(* CODESYS project Warehouse_Final_Plc.project
   Company: ifm electronic
   Description: Project template with CR711S configured 2.25MByte Standard 2.25MByte Safety
   Title: ifmCR711S_TemplateProject
   Version: 2.4.10.0

Project tree, tasks and I/O mapping:
  StandardPLC : CR711S Standard, ifm electronic, order no. CR711S, version 3.2.0.0
    application Application
      libraries: ifmR360-3, 1.1.1.0 (ifm electronic); Util, * (System); Standard, * (System); CR711S IOWrapper, 1.0.4.9 (ifm electronic); CAA CiA 405, 3.5.8.0 (CAA Technical Workgroup)
      task Task (cyclic, interval t#10ms, priority 0) calls PLC_PRG
      global variables inc1
      EVC
      program CR711S_Config [ST]: config_outputs, config_outgroups, config_inputs
      trace Trace (task Task): PLC_PRG.iSlopeLat, PLC_PRG.iSlopeLong
      program PLC_PRG [ST]
      visualisation Visualization
      program Inclination_logic [ST]
      program Temp_Logic [ST]
      program CAN_INIT [ST]
      program CAN_TX [FBD]
      trace Trace_1 (task ): Temp_Logic.TEMPval
      visualisation Visualization_1
      program test [FBD]
    HMI : HMI, ifm electronic, version 3.2.0.0
      User_LEDs : User_LEDs, ifm electronic, version 3.2.0.0
          input  UserLED0_I : LED_IEC_B_INPUT_MAPPING_TYPE  // UserLED0_I
          input  UserLED1_I : LED_IEC_B_INPUT_MAPPING_TYPE  // UserLED1_I
          input  UserLED2_I : LED_IEC_B_INPUT_MAPPING_TYPE  // UserLED2_I
          input  UserLED3_I : LED_IEC_B_INPUT_MAPPING_TYPE  // UserLED3_I
          output UserLED0_Q : LED_IEC_B_OUTPUT_MAPPING_TYPE  // User LED 0
          output UserLED1_Q : LED_IEC_B_OUTPUT_MAPPING_TYPE  // User LED 1
          output UserLED2_Q : LED_IEC_B_OUTPUT_MAPPING_TYPE  // User LED 2
          output UserLED3_Q : LED_IEC_B_OUTPUT_MAPPING_TYPE  // User LED 3
    Local_IO : Local_IO, ifm electronic, version 3.2.0.0
      System_Inputs : System_Inputs, ifm electronic, version 3.2.0.0
          input  VBB30 : IN_SYSTEM_VOLTAGE_INPUT_MAPPING_TYPE  // VBB30
          input  VBB15 : IN_SYSTEM_VOLTAGE_INPUT_MAPPING_TYPE  // VBB15
          input  TemperatureBoard0 : IN_TEMPERATURE_INPUT_MAPPING_TYPE  // TemperatureBoard0
          input  TemperatureChip0 : IN_TEMPERATURE_INPUT_MAPPING_TYPE  // TemperatureChip0
      Inputs : Inputs, ifm electronic, version 3.2.0.0
          input  IN0100_I : IN_MULTIFUNCTION_A_INPUT_MAPPING_TYPE  // IN0100_I
          input  IN0101_I : IN_MULTIFUNCTION_A_INPUT_MAPPING_TYPE  // IN0101_I
          input  IN0102_I : IN_MULTIFUNCTION_A_INPUT_MAPPING_TYPE  // IN0102_I
          input  IN0103_I : IN_MULTIFUNCTION_A_INPUT_MAPPING_TYPE  // IN0103_I
          input  IN0200_I : IN_MULTIFUNCTION_A_INPUT_MAPPING_TYPE  // IN0200_I
          input  IN0201_I : IN_MULTIFUNCTION_A_INPUT_MAPPING_TYPE  // IN0201_I
          input  IN0202_I : IN_MULTIFUNCTION_A_INPUT_MAPPING_TYPE  // IN0202_I
          input  IN0203_I : IN_MULTIFUNCTION_A_INPUT_MAPPING_TYPE  // IN0203_I
          input  IN0600_I : IN_MULTIFUNCTION_A_INPUT_MAPPING_TYPE  // IN0600_I
          input  IN0601_I : IN_MULTIFUNCTION_A_INPUT_MAPPING_TYPE  // IN0601_I
          input  IN0602_I : IN_MULTIFUNCTION_A_INPUT_MAPPING_TYPE  // IN0602_I
          input  IN0603_I : IN_MULTIFUNCTION_A_INPUT_MAPPING_TYPE  // IN0603_I
          input  IN0700_I : IN_MULTIFUNCTION_A_INPUT_MAPPING_TYPE  // IN0700_I
          input  IN0701_I : IN_MULTIFUNCTION_A_INPUT_MAPPING_TYPE  // IN0701_I
          input  IN0702_I : IN_MULTIFUNCTION_A_INPUT_MAPPING_TYPE  // IN0702_I
          input  IN0703_I : IN_MULTIFUNCTION_A_INPUT_MAPPING_TYPE  // IN0703_I
          input  IN0400_I : IN_RESISTOR_A_INPUT_MAPPING_TYPE  // IN0400_I
          input  IN0401_I : IN_RESISTOR_A_INPUT_MAPPING_TYPE  // IN0401_I
          input  IN0900_I : IN_RESISTOR_A_INPUT_MAPPING_TYPE  // IN0900_I
          input  IN0901_I : IN_RESISTOR_A_INPUT_MAPPING_TYPE  // IN0901_I
          input  IN0300_I : IN_DIGITAL_B_INPUT_MAPPING_TYPE  // IN0300_I
          input  IN0301_I : IN_DIGITAL_B_INPUT_MAPPING_TYPE  // IN0301_I
          input  IN0800_I : IN_DIGITAL_B_INPUT_MAPPING_TYPE  // IN0800_I
          input  IN0801_I : IN_DIGITAL_B_INPUT_MAPPING_TYPE  // IN0801_I
          input  COM_RESET_I : IN_COMMUNICATION_RESET_INPUT_MAPPING_TYPE  // COM_RESET_I
          input  IN0000_I : IN_FREQUENCY_B_CHANNEL_A_INPUT_MAPPING_TYPE  // IN0000_I
          input  IN0002_I : IN_FREQUENCY_B_CHANNEL_A_INPUT_MAPPING_TYPE  // IN0002_I
          input  IN0500_I : IN_FREQUENCY_B_CHANNEL_A_INPUT_MAPPING_TYPE  // IN0500_I
          input  IN0502_I : IN_FREQUENCY_B_CHANNEL_A_INPUT_MAPPING_TYPE  // IN0502_I
          input  IN0001_I : IN_FREQUENCY_B_CHANNEL_B_INPUT_MAPPING_TYPE  // IN0001_I
          input  IN0003_I : IN_FREQUENCY_B_CHANNEL_B_INPUT_MAPPING_TYPE  // IN0003_I
          input  IN0501_I : IN_FREQUENCY_B_CHANNEL_B_INPUT_MAPPING_TYPE  // IN0501_I
          input  IN0503_I : IN_FREQUENCY_B_CHANNEL_B_INPUT_MAPPING_TYPE  // IN0503_I
      Outputs : Outputs, ifm electronic, version 3.2.0.0
          input  OUT0006_I : OUT_PWM_40_BRIDGE_A_INPUT_MAPPING_TYPE  // OUT0006_I
          input  OUT0106_I : OUT_PWM_40_BRIDGE_A_INPUT_MAPPING_TYPE  // OUT0106_I
          input  OUT0206_I : OUT_PWM_40_BRIDGE_A_INPUT_MAPPING_TYPE  // OUT0206_I
          input  OUT0008_I : OUT_PWM_40_A_INPUT_MAPPING_TYPE  // OUT0008_I
          input  OUT0108_I : OUT_PWM_40_A_INPUT_MAPPING_TYPE  // OUT0108_I
          input  OUT0208_I : OUT_PWM_40_A_INPUT_MAPPING_TYPE  // OUT0208_I
          input  OUT0000_I : OUT_PWM_25_A_INPUT_MAPPING_TYPE  // OUT0000_I
          input  OUT0002_I : OUT_PWM_25_A_INPUT_MAPPING_TYPE  // OUT0002_I
          input  OUT0004_I : OUT_PWM_25_A_INPUT_MAPPING_TYPE  // OUT0004_I
          input  OUT0100_I : OUT_PWM_25_A_INPUT_MAPPING_TYPE  // OUT0100_I
          input  OUT0102_I : OUT_PWM_25_A_INPUT_MAPPING_TYPE  // OUT0102_I
          input  OUT0104_I : OUT_PWM_25_A_INPUT_MAPPING_TYPE  // OUT0104_I
          input  OUT0200_I : OUT_PWM_25_A_INPUT_MAPPING_TYPE  // OUT0200_I
          input  OUT0202_I : OUT_PWM_25_A_INPUT_MAPPING_TYPE  // OUT0202_I
          input  OUT0204_I : OUT_PWM_25_A_INPUT_MAPPING_TYPE  // OUT0204_I
          input  OUT3001_I : OUT_VOLTAGE_A_INPUT_MAPPING_TYPE  // OUT3001_I
          input  OUT3000_I : OUT_SUPPLY_A_INPUT_MAPPING_TYPE  // OUT3000_I
          input  OUT0001_I : OUT_PWM_25_B_INPUT_MAPPING_TYPE  // OUT0001_I
          input  OUT0003_I : OUT_PWM_25_B_INPUT_MAPPING_TYPE  // OUT0003_I
          input  OUT0005_I : OUT_PWM_25_B_INPUT_MAPPING_TYPE  // OUT0005_I
          input  OUT0101_I : OUT_PWM_25_B_INPUT_MAPPING_TYPE  // OUT0101_I
          input  OUT0103_I : OUT_PWM_25_B_INPUT_MAPPING_TYPE  // OUT0103_I
          input  OUT0105_I : OUT_PWM_25_B_INPUT_MAPPING_TYPE  // OUT0105_I
          input  OUT0201_I : OUT_PWM_25_B_INPUT_MAPPING_TYPE  // OUT0201_I
          input  OUT0203_I : OUT_PWM_25_B_INPUT_MAPPING_TYPE  // OUT0203_I
          input  OUT0205_I : OUT_PWM_25_B_INPUT_MAPPING_TYPE  // OUT0205_I
          input  OUT0007_I : OUT_PWM_40_BRIDGE_A_INPUT_MAPPING_TYPE  // OUT0007_I
          input  OUT0107_I : OUT_PWM_40_BRIDGE_A_INPUT_MAPPING_TYPE  // OUT0107_I
          input  OUT0207_I : OUT_PWM_40_BRIDGE_A_INPUT_MAPPING_TYPE  // OUT0207_I
          output OUT0006_Q : OUT_PWM_40_BRIDGE_A_OUTPUT_MAPPING_TYPE  // OUT0006_Q
          output OUT0106_Q : OUT_PWM_40_BRIDGE_A_OUTPUT_MAPPING_TYPE  // OUT0106_Q
          output OUT0206_Q : OUT_PWM_40_BRIDGE_A_OUTPUT_MAPPING_TYPE  // OUT0206_Q
          output OUT0008_Q : OUT_PWM_40_A_OUTPUT_MAPPING_TYPE  // OUT0008_Q
          output OUT0108_Q : OUT_PWM_40_A_OUTPUT_MAPPING_TYPE  // OUT0108_Q
          output OUT0208_Q : OUT_PWM_40_A_OUTPUT_MAPPING_TYPE  // OUT0208_Q
          output OUT0000_Q : OUT_PWM_25_A_OUTPUT_MAPPING_TYPE  // OUT0000_Q
          output OUT0002_Q : OUT_PWM_25_A_OUTPUT_MAPPING_TYPE  // OUT0002_Q
          output OUT0004_Q : OUT_PWM_25_A_OUTPUT_MAPPING_TYPE  // OUT0004_Q
          output OUT0100_Q : OUT_PWM_25_A_OUTPUT_MAPPING_TYPE  // OUT0100_Q
          output OUT0102_Q : OUT_PWM_25_A_OUTPUT_MAPPING_TYPE  // OUT0102_Q
          output OUT0104_Q : OUT_PWM_25_A_OUTPUT_MAPPING_TYPE  // OUT0104_Q
          output OUT0200_Q : OUT_PWM_25_A_OUTPUT_MAPPING_TYPE  // OUT0200_Q
          output OUT0202_Q : OUT_PWM_25_A_OUTPUT_MAPPING_TYPE  // OUT0202_Q
          output OUT0204_Q : OUT_PWM_25_A_OUTPUT_MAPPING_TYPE  // OUT0204_Q
          output OUT3001_Q : OUT_VOLTAGE_A_OUTPUT_MAPPING_TYPE  // OUT3001_Q
          output OUT3000_Q : OUT_SUPPLY_A_OUTPUT_MAPPING_TYPE  // OUT3000_Q
          output OUT0001_Q : OUT_PWM_25_B_OUTPUT_MAPPING_TYPE  // OUT0001_Q
          output OUT0003_Q : OUT_PWM_25_B_OUTPUT_MAPPING_TYPE  // OUT0003_Q
          output OUT0005_Q : OUT_PWM_25_B_OUTPUT_MAPPING_TYPE  // OUT0005_Q
          output OUT0101_Q : OUT_PWM_25_B_OUTPUT_MAPPING_TYPE  // OUT0101_Q
          output OUT0103_Q : OUT_PWM_25_B_OUTPUT_MAPPING_TYPE  // OUT0103_Q
          output OUT0105_Q : OUT_PWM_25_B_OUTPUT_MAPPING_TYPE  // OUT0105_Q
          output OUT0201_Q : OUT_PWM_25_B_OUTPUT_MAPPING_TYPE  // OUT0201_Q
          output OUT0203_Q : OUT_PWM_25_B_OUTPUT_MAPPING_TYPE  // OUT0203_Q
          output OUT0205_Q : OUT_PWM_25_B_OUTPUT_MAPPING_TYPE  // OUT0205_Q
          output OUT0007_Q : OUT_PWM_40_BRIDGE_A_OUTPUT_MAPPING_TYPE  // OUT0007_Q
          output OUT0107_Q : OUT_PWM_40_BRIDGE_A_OUTPUT_MAPPING_TYPE  // OUT0107_Q
          output OUT0207_Q : OUT_PWM_40_BRIDGE_A_OUTPUT_MAPPING_TYPE  // OUT0207_Q
      System_Outputs : System_Outputs, ifm electronic, version 3.2.0.0
          input  VBB0_SW_I : OUT_GROUP_SWITCH_INPUT_MAPPING_TYPE  // VBB0_SW_I
          input  VBB1_SW_I : OUT_GROUP_SWITCH_INPUT_MAPPING_TYPE  // VBB1_SW_I
          input  VBB2_SW_I : OUT_GROUP_SWITCH_INPUT_MAPPING_TYPE  // VBB2_SW_I
          output VBB0_SW_Q : OUT_GROUP_SWITCH_OUTPUT_MAPPING_TYPE  // VBB0_SW_Q
          output VBB1_SW_Q : OUT_GROUP_SWITCH_OUTPUT_MAPPING_TYPE  // VBB1_SW_Q
          output VBB2_SW_Q : OUT_GROUP_SWITCH_OUTPUT_MAPPING_TYPE  // VBB2_SW_Q
          output SUPPLY_SWITCH_Q : OUT_SYS_SWITCH_OUTPUT_MAPPING_TYPE  // SUPPLY_SWITCH_Q
    Communication : Communication, ifm electronic, version 3.2.0.0
      CAN : CAN, ifm electronic, version 3.2.0.0
        CANbus : CANbus, ifm electronic, version 1.0.1.1
          CANopen_Manager : CANopen_Manager, 3S - Smart Software Solutions GmbH, version 3.5.16.0
              settings: NMT Start All = TRUE; ConfigVersion = 50659584
            JN2100 : JN2100, ifm electornic GmbH, order no. JN2100, version Revision=16#000000AA, FileVersion=1.1, File=JN2100_V2.5.4.eds
                settings: General Options.Optional Device = TRUE; General Options.Reset Node = FALSE; NODEIDSAVED = 10; SDO Timeout = 1000000; PDO_Autoconfig = FALSE; EXPERTSETTINGS = True; Emergency-General Parameters.Emergency COBID = 16#0000008A; Heartbeat-Producer Time = 200; PDO 16#1800.COBID = 16#0000018A; PDO 16#1800.Transmission Type = 16#FE; PDO 16#1800.Event Timer = 50; Process by CANopenManager = TRUE; PDO 16#1801.COBID = 16#0000028A; PDO 16#1801.Transmission Type = 16#01; Process by CANopenManager = TRUE; PDO 16#1802.COBID = 16#0000038A; PDO 16#1802.Transmission Type = 16#01; Process by CANopenManager = TRUE; PDO 16#1803.COBID = 16#0000048A; Process by CANopenManager = TRUE; Slope long16.Subindex = 16#00; Slope lateral16.Subindex = 16#00; Slope long32.Subindex = 16#00; Slope lateral32.Subindex = 16#00; v effektive vector magnitude.Subindex = 16#00; a peak vector magnitude.Subindex = 16#00; a x vector.Subindex = 16#00; a y vector.Subindex = 16#00; a z vector.Subindex = 16#00; SDO List.Set Guardtime.Index = 16#100C; SDO List.Set Guardtime.Subindex = 16#00; SDO List.Set Guardtime.Value = 16#00000000; SDO List.Set Guardtime.Size = 16; SDO List.Set Guardtime.AbortIfError = FALSE; SDO List.Set Guardtime.JumpToLine = FALSE; SDO List.Set Guardtime.Line = 0; SDO List.Set Lifetime.Index = 16#100D; SDO List.Set Lifetime.Subindex = 16#00; SDO List.Set Lifetime.Value = 16#00000000; SDO List.Set Lifetime.Size = 8;
                  SDO List.Set Lifetime.AbortIfError = FALSE; SDO List.Set Lifetime.JumpToLine = FALSE; SDO List.Set Lifetime.Line = 0; SDO List.Set Heartbeat Producer.Index = 16#1017; SDO List.Set Heartbeat Producer.Subindex = 16#00; SDO List.Set Heartbeat Producer.Value = 16#000000C8; SDO List.Set Heartbeat Producer.Size = 16; SDO List.Set Heartbeat Producer.AbortIfError = FALSE; SDO List.Set Heartbeat Producer.JumpToLine = FALSE; SDO List.Set Heartbeat Producer.Line = 0; SDO List.Disable PDO.Index = 16#1800; SDO List.Disable PDO.Subindex = 16#01; SDO List.Disable PDO.Value = 16#8000018A; SDO List.Disable PDO.Size = 32; SDO List.Disable PDO.AbortIfError = FALSE; SDO List.Disable PDO.JumpToLine = FALSE; SDO List.Disable PDO.Line = 0; SDO List.Set transmission type.Index = 16#1800; SDO List.Set transmission type.Subindex = 16#02; SDO List.Set transmission type.Value = 16#FE; SDO List.Set transmission type.Size = 8; SDO List.Set transmission type.AbortIfError = FALSE; SDO List.Set transmission type.JumpToLine = FALSE; SDO List.Set transmission type.Line = 0; SDO List.Set inhibit time.Index = 16#1800; SDO List.Set inhibit time.Subindex = 16#03; SDO List.Set inhibit time.Value = 16#0000; SDO List.Set inhibit time.Size = 16; SDO List.Set inhibit time.AbortIfError = FALSE; SDO List.Set inhibit time.JumpToLine = FALSE; SDO List.Set inhibit time.Line = 0; SDO List.Set event time.Index = 16#1800; SDO List.Set event time.Subindex = 16#05; SDO List.Set event time.Value = 16#0032; SDO List.Set event time.Size = 16; SDO List.Set event time.AbortIfError = FALSE; SDO List.Set event time.JumpToLine = FALSE; SDO List.Set event time.Line = 0; SDO List.Clear pdo mapping.Index = 16#1A00; SDO List.Clear pdo mapping.Subindex = 16#00;
                  SDO List.Clear pdo mapping.Value = 16#0; SDO List.Clear pdo mapping.Size = 8; SDO List.Clear pdo mapping.AbortIfError = FALSE; SDO List.Clear pdo mapping.JumpToLine = FALSE; SDO List.Clear pdo mapping.Line = 0; SDO List.Set Mapping.Index = 16#1A00; SDO List.Set Mapping.Subindex = 16#01; SDO List.Set Mapping.Value = 16#60100010; SDO List.Set Mapping.Size = 32; SDO List.Set Mapping.AbortIfError = FALSE; SDO List.Set Mapping.JumpToLine = FALSE; SDO List.Set Mapping.Line = 0; SDO List.Set Mapping.Index = 16#1A00; SDO List.Set Mapping.Subindex = 16#02; SDO List.Set Mapping.Value = 16#60200010; SDO List.Set Mapping.Size = 32; SDO List.Set Mapping.AbortIfError = FALSE; SDO List.Set Mapping.JumpToLine = FALSE; SDO List.Set Mapping.Line = 0; SDO List.Set number of mappings.Index = 16#1A00; SDO List.Set number of mappings.Subindex = 16#00; SDO List.Set number of mappings.Value = 16#02; SDO List.Set number of mappings.Size = 8; SDO List.Set number of mappings.AbortIfError = FALSE; SDO List.Set number of mappings.JumpToLine = FALSE; SDO List.Set number of mappings.Line = 0; SDO List.Set and enable COB-ID.Index = 16#1800; SDO List.Set and enable COB-ID.Subindex = 16#01; SDO List.Set and enable COB-ID.Value = 16#0000018A; SDO List.Set and enable COB-ID.Size = 32; SDO List.Set and enable COB-ID.AbortIfError = FALSE; SDO List.Set and enable COB-ID.JumpToLine = FALSE; SDO List.Set and enable COB-ID.Line = 0; SDO List.Disable PDO.Index = 16#1801; SDO List.Disable PDO.Subindex = 16#01; SDO List.Disable PDO.Value = 16#8000028A; SDO List.Disable PDO.Size = 32; SDO List.Disable PDO.AbortIfError = FALSE; SDO List.Disable PDO.JumpToLine = FALSE; SDO List.Disable PDO.Line = 0;
                  SDO List.Set transmission type.Index = 16#1801; SDO List.Set transmission type.Subindex = 16#02; SDO List.Set transmission type.Value = 16#01; SDO List.Set transmission type.Size = 8; SDO List.Set transmission type.AbortIfError = FALSE; SDO List.Set transmission type.JumpToLine = FALSE; SDO List.Set transmission type.Line = 0; SDO List.Set inhibit time.Index = 16#1801; SDO List.Set inhibit time.Subindex = 16#03; SDO List.Set inhibit time.Value = 16#0000; SDO List.Set inhibit time.Size = 16; SDO List.Set inhibit time.AbortIfError = FALSE; SDO List.Set inhibit time.JumpToLine = FALSE; SDO List.Set inhibit time.Line = 0; SDO List.Set event time.Index = 16#1801; SDO List.Set event time.Subindex = 16#05; SDO List.Set event time.Value = 16#000A; SDO List.Set event time.Size = 16; SDO List.Set event time.AbortIfError = FALSE; SDO List.Set event time.JumpToLine = FALSE; SDO List.Set event time.Line = 0; SDO List.Clear pdo mapping.Index = 16#1A01; SDO List.Clear pdo mapping.Subindex = 16#00; SDO List.Clear pdo mapping.Value = 16#0; SDO List.Clear pdo mapping.Size = 8; SDO List.Clear pdo mapping.AbortIfError = FALSE; SDO List.Clear pdo mapping.JumpToLine = FALSE; SDO List.Clear pdo mapping.Line = 0; SDO List.Set Mapping.Index = 16#1A01; SDO List.Set Mapping.Subindex = 16#01; SDO List.Set Mapping.Value = 16#61100020; SDO List.Set Mapping.Size = 32; SDO List.Set Mapping.AbortIfError = FALSE; SDO List.Set Mapping.JumpToLine = FALSE; SDO List.Set Mapping.Line = 0; SDO List.Set Mapping.Index = 16#1A01; SDO List.Set Mapping.Subindex = 16#02; SDO List.Set Mapping.Value = 16#61200020; SDO List.Set Mapping.Size = 32; SDO List.Set Mapping.AbortIfError = FALSE;
                  SDO List.Set Mapping.JumpToLine = FALSE; SDO List.Set Mapping.Line = 0; SDO List.Set number of mappings.Index = 16#1A01; SDO List.Set number of mappings.Subindex = 16#00; SDO List.Set number of mappings.Value = 16#02; SDO List.Set number of mappings.Size = 8; SDO List.Set number of mappings.AbortIfError = FALSE; SDO List.Set number of mappings.JumpToLine = FALSE; SDO List.Set number of mappings.Line = 0; SDO List.Set and enable COB-ID.Index = 16#1801; SDO List.Set and enable COB-ID.Subindex = 16#01; SDO List.Set and enable COB-ID.Value = 16#0000028A; SDO List.Set and enable COB-ID.Size = 32; SDO List.Set and enable COB-ID.AbortIfError = FALSE; SDO List.Set and enable COB-ID.JumpToLine = FALSE; SDO List.Set and enable COB-ID.Line = 0; SDO List.Disable PDO.Index = 16#1802; SDO List.Disable PDO.Subindex = 16#01; SDO List.Disable PDO.Value = 16#8000038A; SDO List.Disable PDO.Size = 32; SDO List.Disable PDO.AbortIfError = FALSE; SDO List.Disable PDO.JumpToLine = FALSE; SDO List.Disable PDO.Line = 0; SDO List.Set transmission type.Index = 16#1802; SDO List.Set transmission type.Subindex = 16#02; SDO List.Set transmission type.Value = 16#01; SDO List.Set transmission type.Size = 8; SDO List.Set transmission type.AbortIfError = FALSE; SDO List.Set transmission type.JumpToLine = FALSE; SDO List.Set transmission type.Line = 0; SDO List.Set inhibit time.Index = 16#1802; SDO List.Set inhibit time.Subindex = 16#03; SDO List.Set inhibit time.Value = 16#0000; SDO List.Set inhibit time.Size = 16; SDO List.Set inhibit time.AbortIfError = FALSE; SDO List.Set inhibit time.JumpToLine = FALSE; SDO List.Set inhibit time.Line = 0; SDO List.Set event time.Index = 16#1802; SDO List.Set event time.Subindex = 16#05; SDO List.Set event time.Value = 16#000A;
                  SDO List.Set event time.Size = 16; SDO List.Set event time.AbortIfError = FALSE; SDO List.Set event time.JumpToLine = FALSE; SDO List.Set event time.Line = 0; SDO List.Clear pdo mapping.Index = 16#1A02; SDO List.Clear pdo mapping.Subindex = 16#00; SDO List.Clear pdo mapping.Value = 16#0; SDO List.Clear pdo mapping.Size = 8; SDO List.Clear pdo mapping.AbortIfError = FALSE; SDO List.Clear pdo mapping.JumpToLine = FALSE; SDO List.Clear pdo mapping.Line = 0; SDO List.Set Mapping.Index = 16#1A02; SDO List.Set Mapping.Subindex = 16#01; SDO List.Set Mapping.Value = 16#5C100020; SDO List.Set Mapping.Size = 32; SDO List.Set Mapping.AbortIfError = FALSE; SDO List.Set Mapping.JumpToLine = FALSE; SDO List.Set Mapping.Line = 0; SDO List.Set Mapping.Index = 16#1A02; SDO List.Set Mapping.Subindex = 16#02; SDO List.Set Mapping.Value = 16#5C110020; SDO List.Set Mapping.Size = 32; SDO List.Set Mapping.AbortIfError = FALSE; SDO List.Set Mapping.JumpToLine = FALSE; SDO List.Set Mapping.Line = 0; SDO List.Set number of mappings.Index = 16#1A02; SDO List.Set number of mappings.Subindex = 16#00; SDO List.Set number of mappings.Value = 16#02; SDO List.Set number of mappings.Size = 8; SDO List.Set number of mappings.AbortIfError = FALSE; SDO List.Set number of mappings.JumpToLine = FALSE; SDO List.Set number of mappings.Line = 0; SDO List.Set and enable COB-ID.Index = 16#1802; SDO List.Set and enable COB-ID.Subindex = 16#01; SDO List.Set and enable COB-ID.Value = 16#0000038A; SDO List.Set and enable COB-ID.Size = 32; SDO List.Set and enable COB-ID.AbortIfError = FALSE; SDO List.Set and enable COB-ID.JumpToLine = FALSE; SDO List.Set and enable COB-ID.Line = 0; SDO List.Disable PDO.Index = 16#1803;
                  SDO List.Disable PDO.Subindex = 16#01; SDO List.Disable PDO.Value = 16#8000048A; SDO List.Disable PDO.Size = 32; SDO List.Disable PDO.AbortIfError = FALSE; SDO List.Disable PDO.JumpToLine = FALSE; SDO List.Disable PDO.Line = 0; SDO List.Set transmission type.Index = 16#1803; SDO List.Set transmission type.Subindex = 16#02; SDO List.Set transmission type.Value = 16#FF; SDO List.Set transmission type.Size = 8; SDO List.Set transmission type.AbortIfError = FALSE; SDO List.Set transmission type.JumpToLine = FALSE; SDO List.Set transmission type.Line = 0; SDO List.Set inhibit time.Index = 16#1803; SDO List.Set inhibit time.Subindex = 16#03; SDO List.Set inhibit time.Value = 16#0000; SDO List.Set inhibit time.Size = 16; SDO List.Set inhibit time.AbortIfError = FALSE; SDO List.Set inhibit time.JumpToLine = FALSE; SDO List.Set inhibit time.Line = 0; SDO List.Set event time.Index = 16#1803; SDO List.Set event time.Subindex = 16#05; SDO List.Set event time.Value = 16#000A; SDO List.Set event time.Size = 16; SDO List.Set event time.AbortIfError = FALSE; SDO List.Set event time.JumpToLine = FALSE; SDO List.Set event time.Line = 0; SDO List.Clear pdo mapping.Index = 16#1A03; SDO List.Clear pdo mapping.Subindex = 16#00; SDO List.Clear pdo mapping.Value = 16#0; SDO List.Clear pdo mapping.Size = 8; SDO List.Clear pdo mapping.AbortIfError = FALSE; SDO List.Clear pdo mapping.JumpToLine = FALSE; SDO List.Clear pdo mapping.Line = 0; SDO List.Set Mapping.Index = 16#1A03; SDO List.Set Mapping.Subindex = 16#01; SDO List.Set Mapping.Value = 16#5D100010; SDO List.Set Mapping.Size = 32; SDO List.Set Mapping.AbortIfError = FALSE; SDO List.Set Mapping.JumpToLine = FALSE;
                  SDO List.Set Mapping.Line = 0; SDO List.Set Mapping.Index = 16#1A03; SDO List.Set Mapping.Subindex = 16#02; SDO List.Set Mapping.Value = 16#5D110010; SDO List.Set Mapping.Size = 32; SDO List.Set Mapping.AbortIfError = FALSE; SDO List.Set Mapping.JumpToLine = FALSE; SDO List.Set Mapping.Line = 0; SDO List.Set Mapping.Index = 16#1A03; SDO List.Set Mapping.Subindex = 16#03; SDO List.Set Mapping.Value = 16#5D120010; SDO List.Set Mapping.Size = 32; SDO List.Set Mapping.AbortIfError = FALSE; SDO List.Set Mapping.JumpToLine = FALSE; SDO List.Set Mapping.Line = 0; SDO List.Set number of mappings.Index = 16#1A03; SDO List.Set number of mappings.Subindex = 16#00; SDO List.Set number of mappings.Value = 16#03; SDO List.Set number of mappings.Size = 8; SDO List.Set number of mappings.AbortIfError = FALSE; SDO List.Set number of mappings.JumpToLine = FALSE; SDO List.Set number of mappings.Line = 0; SDO List.Set and enable COB-ID.Index = 16#1803; SDO List.Set and enable COB-ID.Subindex = 16#01; SDO List.Set and enable COB-ID.Value = 16#0000048A; SDO List.Set and enable COB-ID.Size = 32; SDO List.Set and enable COB-ID.AbortIfError = FALSE; SDO List.Set and enable COB-ID.JumpToLine = FALSE; SDO List.Set and enable COB-ID.Line = 0; ConfigVersion = 50659584
                input  Application.PLC_PRG.iSlopeLong : INT  // Slope long16
                input  Application.PLC_PRG.iSlopeLat : INT  // Slope lateral16
                unmapped channels: Slope long32, Slope lateral32, v effektive vector magnitude, a peak vector magnitude, a x vector, a y vector, a z vector
      Ethernet : Ethernet, ifm electronic, version 3.2.0.0
  SafetyPLC : CR711S SIL2, ifm electronic, order no. CR711S, version 3.2.0.0
    application Application
      libraries: ifmR360-3, * (ifm electronic)
      task Task (cyclic, interval t#10ms, priority 1, watchdog t#8ms x 1) calls PLC_PRG
      program PLC_PRG [ST]
      global variables EVL
    HMI : HMI, ifm electronic, version 3.2.0.0
      User_LEDs : User_LEDs, ifm electronic, version 3.2.0.0
          input  UserLED0_I : LED_IEC_B_INPUT_MAPPING_TYPE  // UserLED0_I
          input  UserLED1_I : LED_IEC_B_INPUT_MAPPING_TYPE  // UserLED1_I
          input  UserLED2_I : LED_IEC_B_INPUT_MAPPING_TYPE  // UserLED2_I
          input  UserLED3_I : LED_IEC_B_INPUT_MAPPING_TYPE  // UserLED3_I
          output UserLED0_Q : LED_IEC_B_OUTPUT_MAPPING_TYPE  // User LED 0
          output UserLED1_Q : LED_IEC_B_OUTPUT_MAPPING_TYPE  // User LED 1
          output UserLED2_Q : LED_IEC_B_OUTPUT_MAPPING_TYPE  // User LED 2
          output UserLED3_Q : LED_IEC_B_OUTPUT_MAPPING_TYPE  // User LED 3
    Local_IO : Local_IO, ifm electronic, version 3.2.0.0
      System_Outputs : System_Outputs, ifm electronic, version 3.2.0.0
          input  VBB0_SW_I : OUT_GROUP_SWITCH_INPUT_MAPPING_TYPE  // VBB0_SW_I
          input  VBB1_SW_I : OUT_GROUP_SWITCH_INPUT_MAPPING_TYPE  // VBB1_SW_I
          input  VBB2_SW_I : OUT_GROUP_SWITCH_INPUT_MAPPING_TYPE  // VBB2_SW_I
          output VBB0_SW_Q : OUT_GROUP_SWITCH_OUTPUT_MAPPING_TYPE  // VBB0_SW_Q
          output VBB1_SW_Q : OUT_GROUP_SWITCH_OUTPUT_MAPPING_TYPE  // VBB1_SW_Q
          output VBB2_SW_Q : OUT_GROUP_SWITCH_OUTPUT_MAPPING_TYPE  // VBB2_SW_Q
          output SUPPLY_SWITCH_Q : OUT_SYS_SWITCH_OUTPUT_MAPPING_TYPE  // SUPPLY_SWITCH_Q
      Outputs : Outputs, ifm electronic, version 3.2.0.0
          input  OUT0006_I : OUT_PWM_40_BRIDGE_A_INPUT_MAPPING_TYPE  // OUT0006_I
          input  OUT0106_I : OUT_PWM_40_BRIDGE_A_INPUT_MAPPING_TYPE  // OUT0106_I
          input  OUT0206_I : OUT_PWM_40_BRIDGE_A_INPUT_MAPPING_TYPE  // OUT0206_I
          input  OUT0008_I : OUT_PWM_40_A_INPUT_MAPPING_TYPE  // OUT0008_I
          input  OUT0108_I : OUT_PWM_40_A_INPUT_MAPPING_TYPE  // OUT0108_I
          input  OUT0208_I : OUT_PWM_40_A_INPUT_MAPPING_TYPE  // OUT0208_I
          input  OUT0000_I : OUT_PWM_25_A_INPUT_MAPPING_TYPE  // OUT0000_I
          input  OUT0002_I : OUT_PWM_25_A_INPUT_MAPPING_TYPE  // OUT0002_I
          input  OUT0004_I : OUT_PWM_25_A_INPUT_MAPPING_TYPE  // OUT0004_I
          input  OUT0100_I : OUT_PWM_25_A_INPUT_MAPPING_TYPE  // OUT0100_I
          input  OUT0102_I : OUT_PWM_25_A_INPUT_MAPPING_TYPE  // OUT0102_I
          input  OUT0104_I : OUT_PWM_25_A_INPUT_MAPPING_TYPE  // OUT0104_I
          input  OUT0200_I : OUT_PWM_25_A_INPUT_MAPPING_TYPE  // OUT0200_I
          input  OUT0202_I : OUT_PWM_25_A_INPUT_MAPPING_TYPE  // OUT0202_I
          input  OUT0204_I : OUT_PWM_25_A_INPUT_MAPPING_TYPE  // OUT0204_I
          input  OUT3001_I : OUT_VOLTAGE_A_INPUT_MAPPING_TYPE  // OUT3001_I
          input  OUT3000_I : OUT_SUPPLY_A_INPUT_MAPPING_TYPE  // OUT3000_I
          input  OUT0001_I : OUT_PWM_25_B_INPUT_MAPPING_TYPE  // OUT0001_I
          input  OUT0003_I : OUT_PWM_25_B_INPUT_MAPPING_TYPE  // OUT0003_I
          input  OUT0005_I : OUT_PWM_25_B_INPUT_MAPPING_TYPE  // OUT0005_I
          input  OUT0101_I : OUT_PWM_25_B_INPUT_MAPPING_TYPE  // OUT0101_I
          input  OUT0103_I : OUT_PWM_25_B_INPUT_MAPPING_TYPE  // OUT0103_I
          input  OUT0105_I : OUT_PWM_25_B_INPUT_MAPPING_TYPE  // OUT0105_I
          input  OUT0201_I : OUT_PWM_25_B_INPUT_MAPPING_TYPE  // OUT0201_I
          input  OUT0203_I : OUT_PWM_25_B_INPUT_MAPPING_TYPE  // OUT0203_I
          input  OUT0205_I : OUT_PWM_25_B_INPUT_MAPPING_TYPE  // OUT0205_I
          input  OUT0007_I : OUT_PWM_40_BRIDGE_A_INPUT_MAPPING_TYPE  // OUT0007_I
          input  OUT0107_I : OUT_PWM_40_BRIDGE_A_INPUT_MAPPING_TYPE  // OUT0107_I
          input  OUT0207_I : OUT_PWM_40_BRIDGE_A_INPUT_MAPPING_TYPE  // OUT0207_I
          output OUT0006_Q : OUT_PWM_40_BRIDGE_A_OUTPUT_MAPPING_TYPE  // OUT0006_Q
          output OUT0106_Q : OUT_PWM_40_BRIDGE_A_OUTPUT_MAPPING_TYPE  // OUT0106_Q
          output OUT0206_Q : OUT_PWM_40_BRIDGE_A_OUTPUT_MAPPING_TYPE  // OUT0206_Q
          output OUT0008_Q : OUT_PWM_40_A_OUTPUT_MAPPING_TYPE  // OUT0008_Q
          output OUT0108_Q : OUT_PWM_40_A_OUTPUT_MAPPING_TYPE  // OUT0108_Q
          output OUT0208_Q : OUT_PWM_40_A_OUTPUT_MAPPING_TYPE  // OUT0208_Q
          output OUT0000_Q : OUT_PWM_25_A_OUTPUT_MAPPING_TYPE  // OUT0000_Q
          output OUT0002_Q : OUT_PWM_25_A_OUTPUT_MAPPING_TYPE  // OUT0002_Q
          output OUT0004_Q : OUT_PWM_25_A_OUTPUT_MAPPING_TYPE  // OUT0004_Q
          output OUT0100_Q : OUT_PWM_25_A_OUTPUT_MAPPING_TYPE  // OUT0100_Q
          output OUT0102_Q : OUT_PWM_25_A_OUTPUT_MAPPING_TYPE  // OUT0102_Q
          output OUT0104_Q : OUT_PWM_25_A_OUTPUT_MAPPING_TYPE  // OUT0104_Q
          output OUT0200_Q : OUT_PWM_25_A_OUTPUT_MAPPING_TYPE  // OUT0200_Q
          output OUT0202_Q : OUT_PWM_25_A_OUTPUT_MAPPING_TYPE  // OUT0202_Q
          output OUT0204_Q : OUT_PWM_25_A_OUTPUT_MAPPING_TYPE  // OUT0204_Q
          output OUT3001_Q : OUT_VOLTAGE_A_OUTPUT_MAPPING_TYPE  // OUT3001_Q
          output OUT3000_Q : OUT_SUPPLY_A_OUTPUT_MAPPING_TYPE  // OUT3000_Q
          output OUT0001_Q : OUT_PWM_25_B_OUTPUT_MAPPING_TYPE  // OUT0001_Q
          output OUT0003_Q : OUT_PWM_25_B_OUTPUT_MAPPING_TYPE  // OUT0003_Q
          output OUT0005_Q : OUT_PWM_25_B_OUTPUT_MAPPING_TYPE  // OUT0005_Q
          output OUT0101_Q : OUT_PWM_25_B_OUTPUT_MAPPING_TYPE  // OUT0101_Q
          output OUT0103_Q : OUT_PWM_25_B_OUTPUT_MAPPING_TYPE  // OUT0103_Q
          output OUT0105_Q : OUT_PWM_25_B_OUTPUT_MAPPING_TYPE  // OUT0105_Q
          output OUT0201_Q : OUT_PWM_25_B_OUTPUT_MAPPING_TYPE  // OUT0201_Q
          output OUT0203_Q : OUT_PWM_25_B_OUTPUT_MAPPING_TYPE  // OUT0203_Q
          output OUT0205_Q : OUT_PWM_25_B_OUTPUT_MAPPING_TYPE  // OUT0205_Q
          output OUT0007_Q : OUT_PWM_40_BRIDGE_A_OUTPUT_MAPPING_TYPE  // OUT0007_Q
          output OUT0107_Q : OUT_PWM_40_BRIDGE_A_OUTPUT_MAPPING_TYPE  // OUT0107_Q
          output OUT0207_Q : OUT_PWM_40_BRIDGE_A_OUTPUT_MAPPING_TYPE  // OUT0207_Q
      System_Inputs : System_Inputs, ifm electronic, version 3.2.0.0
          input  VBB30 : IN_SYSTEM_VOLTAGE_INPUT_MAPPING_TYPE  // VBB30
          input  VBB15 : IN_SYSTEM_VOLTAGE_INPUT_MAPPING_TYPE  // VBB15
          input  TemperatureBoard0 : IN_TEMPERATURE_INPUT_MAPPING_TYPE  // TemperatureBoard0
          input  TemperatureChip0 : IN_TEMPERATURE_INPUT_MAPPING_TYPE  // TemperatureChip0
      Inputs : Inputs, ifm electronic, version 3.2.0.0
          input  IN0100_I : IN_MULTIFUNCTION_A_INPUT_MAPPING_TYPE  // IN0100_I
          input  IN0101_I : IN_MULTIFUNCTION_A_INPUT_MAPPING_TYPE  // IN0101_I
          input  IN0102_I : IN_MULTIFUNCTION_A_INPUT_MAPPING_TYPE  // IN0102_I
          input  IN0103_I : IN_MULTIFUNCTION_A_INPUT_MAPPING_TYPE  // IN0103_I
          input  IN0200_I : IN_MULTIFUNCTION_A_INPUT_MAPPING_TYPE  // IN0200_I
          input  IN0201_I : IN_MULTIFUNCTION_A_INPUT_MAPPING_TYPE  // IN0201_I
          input  IN0202_I : IN_MULTIFUNCTION_A_INPUT_MAPPING_TYPE  // IN0202_I
          input  IN0203_I : IN_MULTIFUNCTION_A_INPUT_MAPPING_TYPE  // IN0203_I
          input  IN0600_I : IN_MULTIFUNCTION_A_INPUT_MAPPING_TYPE  // IN0600_I
          input  IN0601_I : IN_MULTIFUNCTION_A_INPUT_MAPPING_TYPE  // IN0601_I
          input  IN0602_I : IN_MULTIFUNCTION_A_INPUT_MAPPING_TYPE  // IN0602_I
          input  IN0603_I : IN_MULTIFUNCTION_A_INPUT_MAPPING_TYPE  // IN0603_I
          input  IN0700_I : IN_MULTIFUNCTION_A_INPUT_MAPPING_TYPE  // IN0700_I
          input  IN0701_I : IN_MULTIFUNCTION_A_INPUT_MAPPING_TYPE  // IN0701_I
          input  IN0702_I : IN_MULTIFUNCTION_A_INPUT_MAPPING_TYPE  // IN0702_I
          input  IN0703_I : IN_MULTIFUNCTION_A_INPUT_MAPPING_TYPE  // IN0703_I
          input  IN0400_I : IN_RESISTOR_A_INPUT_MAPPING_TYPE  // IN0400_I
          input  IN0401_I : IN_RESISTOR_A_INPUT_MAPPING_TYPE  // IN0401_I
          input  IN0900_I : IN_RESISTOR_A_INPUT_MAPPING_TYPE  // IN0900_I
          input  IN0901_I : IN_RESISTOR_A_INPUT_MAPPING_TYPE  // IN0901_I
          input  IN0300_I : IN_DIGITAL_B_INPUT_MAPPING_TYPE  // IN0300_I
          input  IN0301_I : IN_DIGITAL_B_INPUT_MAPPING_TYPE  // IN0301_I
          input  IN0800_I : IN_DIGITAL_B_INPUT_MAPPING_TYPE  // IN0800_I
          input  IN0801_I : IN_DIGITAL_B_INPUT_MAPPING_TYPE  // IN0801_I
          input  COM_RESET_I : IN_COMMUNICATION_RESET_INPUT_MAPPING_TYPE  // COM_RESET_I
          input  IN0000_I : IN_FREQUENCY_B_CHANNEL_A_INPUT_MAPPING_TYPE  // IN0000_I
          input  IN0002_I : IN_FREQUENCY_B_CHANNEL_A_INPUT_MAPPING_TYPE  // IN0002_I
          input  IN0500_I : IN_FREQUENCY_B_CHANNEL_A_INPUT_MAPPING_TYPE  // IN0500_I
          input  IN0502_I : IN_FREQUENCY_B_CHANNEL_A_INPUT_MAPPING_TYPE  // IN0502_I
          input  IN0001_I : IN_FREQUENCY_B_CHANNEL_B_INPUT_MAPPING_TYPE  // IN0001_I
          input  IN0003_I : IN_FREQUENCY_B_CHANNEL_B_INPUT_MAPPING_TYPE  // IN0003_I
          input  IN0501_I : IN_FREQUENCY_B_CHANNEL_B_INPUT_MAPPING_TYPE  // IN0501_I
          input  IN0503_I : IN_FREQUENCY_B_CHANNEL_B_INPUT_MAPPING_TYPE  // IN0503_I
    Communication : Communication, ifm electronic, version 3.2.0.0
      Ethernet : Ethernet, ifm electronic, version 3.2.0.0
      CAN : CAN, ifm electronic, version 3.2.0.0
  CR711S : CR711S, ifm electronic, order no. CR711S, version 3.2.0.0
  libraries: VisuSymbols, 3.5.10.0 (System)
  text list GlobalTextList
*)

// StandardPLC/Application/inc1
{attribute 'qualified_only'}
VAR_GLOBAL
	array1:ARRAY [0..7] OF INT;
	
END_VAR

// SafetyPLC/Application/EVL
(* THIS EVL IS AUTOGENERATED. DO NOT MODIFY THESE ATTRIBUTES. *)
{attribute 'location' := '16#800' }
{attribute 'linkalways'}
{attribute 'qualified_only'}
VAR_GLOBAL

END_VAR

// SafetyPLC/Application/PLC_PRG
PROGRAM PLC_PRG
VAR

END_VAR

END_PROGRAM

// StandardPLC/Application/PLC_PRG
PROGRAM PLC_PRG
VAR
  
	
	Inclination_Long: INT;
	Inclination_Lat: INT;
	Rounded_Temp        : INT;
	
// Trigger for the hooter
    // Data structure for inclination data
     // Data array for inclination
	iSlopeLong: INT;
	iSlopeLat: INT;
	rawAnalogTemp : INT;  
	Temperature_Celsius: INT;
END_VAR
(*
IOWrapper V1.0.4.4
ifm ecomatic gmbh - VNC - pp 

The licence free software is of average quality and suitable for normal use on common personal
computers. According to the present state of software technology no guarantee can be
assumed for the correct operation or absence of computer viruses nor for the removal of any
fault which may occur. In case of an incorrect program ifm electronic gmbh cannot be held
liable for cost incurred at the customer (e.g. maintenance, repair or rectification of faults).
The exclusion does not apply to damage for which liability is mandatory according to peremptory
legal provisions. Copyright by ifm electronic gmbh, Essen. No copies may be made without the
written permission of ifm electronic gmbh. This also goes for printing images or text for business
use. We reserve the right to make technical alterations.
*)

CR711S_Config(); 			//IO Configuration

IOWrapper.READ_INPUTS(); 	//Call IOWrapper Main Program and Read Data from Inputs   
CAN_INIT();
CAN_TX();
						//Put your Application program here 
Inclination_logic();

inc1.array1[0] := iSlopeLong;
inc1.array1[1] := iSlopeLat;


	
Temp_Logic();

//test();
IOWrapper.WRITE_OUTPUTS();	//Call IOWrapper Main Program and Write Data to Outputs

END_PROGRAM

// StandardPLC/Application/CR711S_Config
PROGRAM CR711S_Config
VAR_INPUT
END_VAR
(*
IOWrapper V1.4.2.3
ifm ecomatic - VNC - pp 

The licence free software is of average quality and suitable for normal use on common personal
computers. According to the present state of software technology no guarantee can be
assumed for the correct operation or absence of computer viruses nor for the removal of any
fault which may occur. In case of an incorrect program ifm electronic gmbh cannot be held
liable for cost incurred at the customer (e.g. maintenance, repair or rectification of faults).
The exclusion does not apply to damage for which liability is mandatory according to peremptory
legal provisions. Copyright by ifm electronic gmbh, Essen. No copies may be made without the
written permission of ifm electronic gmbh. This also goes for printing images or text for business
use. We reserve the right to make technical alterations.
*)

(* IO Configuration*)
config_inputs();
config_outputs();
config_outgroups();

ACTION config_outputs:
(* Output Mode Configuration *) 
(* Group 0 *)
OUT0000.CONFIG.MONITOR				(FILTER_OUTPUT.UNCHANGED);
OUT0001.CONFIG.OUT_DIGITAL_CSO			(FILTER_OUTPUT.UNCHANGED);
OUT0002.CONFIG.OUT_DIGITAL_CSO				(FILTER_OUTPUT.UNCHANGED);
OUT0003.CONFIG.OUT_DIGITAL_CSO				(FILTER_OUTPUT.UNCHANGED);
OUT0004.CONFIG.MONITOR				(FILTER_OUTPUT.UNCHANGED);
OUT0005.CONFIG.MONITOR				(FILTER_OUTPUT.UNCHANGED);
OUT0006.CONFIG.OUT_HBRIDGE_A				(Temp_Logic.uiFrequency,ifmOUTHBridge.MODE_BRAKE.BRAKE_OFF,T#0MS);
OUT0007.CONFIG.OUT_HBRIDGE_B			();
OUT0008.CONFIG.MONITOR				(FILTER_OUTPUT.UNCHANGED);
(* Group 1 *)         				    		
OUT0100.CONFIG.MONITOR			(FILTER_OUTPUT.UNCHANGED);
OUT0101.CONFIG.MONITOR				(FILTER_OUTPUT.UNCHANGED);
OUT0102.CONFIG.MONITOR				(FILTER_OUTPUT.UNCHANGED);
OUT0103.CONFIG.MONITOR				(FILTER_OUTPUT.UNCHANGED);
OUT0104.CONFIG.MONITOR				(FILTER_OUTPUT.UNCHANGED);
OUT0105.CONFIG.MONITOR				(FILTER_OUTPUT.UNCHANGED);
OUT0106.CONFIG.MONITOR				(FILTER_OUTPUT.UNCHANGED);
OUT0107.CONFIG.MONITOR				(FILTER_OUTPUT.UNCHANGED);
OUT0108.CONFIG.MONITOR				(FILTER_OUTPUT.UNCHANGED);
(* Group 2 *)         				    		
OUT0200.CONFIG.MONITOR				(FILTER_OUTPUT.UNCHANGED);
OUT0201.CONFIG.MONITOR				(FILTER_OUTPUT.UNCHANGED);
OUT0202.CONFIG.MONITOR				(FILTER_OUTPUT.UNCHANGED);
OUT0203.CONFIG.MONITOR				(FILTER_OUTPUT.UNCHANGED);
OUT0204.CONFIG.MONITOR				(FILTER_OUTPUT.UNCHANGED);
OUT0205.CONFIG.MONITOR				(FILTER_OUTPUT.UNCHANGED);
OUT0206.CONFIG.MONITOR				(FILTER_OUTPUT.UNCHANGED);
OUT0207.CONFIG.MONITOR				(FILTER_OUTPUT.UNCHANGED);
OUT0208.CONFIG.MONITOR				(FILTER_OUTPUT.UNCHANGED);
(* Output SensorSupply and Analogue *)      				           				
OUT3000.CONFIG.MONITOR				(FILTER_OUTPUT.UNCHANGED);
OUT3001.CONFIG.MONITOR				(FILTER_OUTPUT.UNCHANGED);

(* Diagnostic and Protection Configuration *) 
(* Group 0 *)
OUT0000.CONFIG.SET_DIAG_LVL_PROT	(0, 2500, 100, eDIAG_PROT_MODE.DIAG_PROT);
OUT0001.CONFIG.SET_DIAG_LVL_PROT	(0, 2500, 100, eDIAG_PROT_MODE.DIAG_PROT);
OUT0002.CONFIG.SET_DIAG_LVL_PROT	(0, 2500, 100, eDIAG_PROT_MODE.DIAG_PROT);
OUT0003.CONFIG.SET_DIAG_LVL_PROT	(0, 2500, 100, eDIAG_PROT_MODE.DIAG_PROT);
OUT0004.CONFIG.SET_DIAG_LVL_PROT	(0, 2500, 100, eDIAG_PROT_MODE.DIAG_PROT);
OUT0005.CONFIG.SET_DIAG_LVL_PROT	(0, 2500, 100, eDIAG_PROT_MODE.DIAG_PROT);
OUT0006.CONFIG.SET_DIAG_LVL_PROT	(0, 4000, 100, eDIAG_PROT_MODE.DIAG_PROT);
OUT0007.CONFIG.SET_DIAG_LVL_PROT	(0, 4000, 100, eDIAG_PROT_MODE.DIAG_PROT);
OUT0008.CONFIG.SET_DIAG_LVL_PROT	(0, 4000, 100, eDIAG_PROT_MODE.DIAG_PROT);
(* Group 1 *)                                       
OUT0100.CONFIG.SET_DIAG_LVL_PROT	(0, 2500, 100, eDIAG_PROT_MODE.DIAG_PROT);
OUT0101.CONFIG.SET_DIAG_LVL_PROT	(0, 2500, 100, eDIAG_PROT_MODE.DIAG_PROT);
OUT0102.CONFIG.SET_DIAG_LVL_PROT	(0, 2500, 100, eDIAG_PROT_MODE.DIAG_PROT);
OUT0103.CONFIG.SET_DIAG_LVL_PROT	(0, 2500, 100, eDIAG_PROT_MODE.DIAG_PROT);
OUT0104.CONFIG.SET_DIAG_LVL_PROT	(0, 2500, 100, eDIAG_PROT_MODE.DIAG_PROT);
OUT0105.CONFIG.SET_DIAG_LVL_PROT	(0, 2500, 100, eDIAG_PROT_MODE.DIAG_PROT);
OUT0106.CONFIG.SET_DIAG_LVL_PROT	(0, 4000, 100, eDIAG_PROT_MODE.DIAG_PROT);
OUT0107.CONFIG.SET_DIAG_LVL_PROT	(0, 4000, 100, eDIAG_PROT_MODE.DIAG_PROT);
OUT0108.CONFIG.SET_DIAG_LVL_PROT	(0, 4000, 100, eDIAG_PROT_MODE.DIAG_PROT);
(* Group 2 *)                                       
OUT0200.CONFIG.SET_DIAG_LVL_PROT	(0, 2500, 100, eDIAG_PROT_MODE.DIAG_PROT);
OUT0201.CONFIG.SET_DIAG_LVL_PROT	(0, 2500, 100, eDIAG_PROT_MODE.DIAG_PROT);
OUT0202.CONFIG.SET_DIAG_LVL_PROT	(0, 2500, 100, eDIAG_PROT_MODE.DIAG_PROT);
OUT0203.CONFIG.SET_DIAG_LVL_PROT	(0, 2500, 100, eDIAG_PROT_MODE.DIAG_PROT);
OUT0204.CONFIG.SET_DIAG_LVL_PROT	(0, 2500, 100, eDIAG_PROT_MODE.DIAG_PROT);
OUT0205.CONFIG.SET_DIAG_LVL_PROT	(0, 2500, 100, eDIAG_PROT_MODE.DIAG_PROT);
OUT0206.CONFIG.SET_DIAG_LVL_PROT	(0, 4000, 100, eDIAG_PROT_MODE.DIAG_PROT);
OUT0207.CONFIG.SET_DIAG_LVL_PROT	(0, 4000, 100, eDIAG_PROT_MODE.DIAG_PROT);
OUT0208.CONFIG.SET_DIAG_LVL_PROT	(0, 4000, 100, eDIAG_PROT_MODE.DIAG_PROT);
END_ACTION

ACTION config_outgroups:
(* Output Group Mode Configuration *) 
OUTGROUP0.CONFIG.MONITOR				(FILTER_OUTPUT_GROUP.UNCHANGED);
OUTGROUP1.CONFIG.MONITOR				(FILTER_OUTPUT_GROUP.UNCHANGED);
OUTGROUP2.CONFIG.MONITOR				(FILTER_OUTPUT_GROUP.UNCHANGED);

(* Diagnostic and Protection Configuration *) 
OUTGROUP0.CONFIG.SET_DIAG_LVL_PROT		(0, 12000, 100, eDIAG_PROT_MODE.DIAG_PROT);
OUTGROUP1.CONFIG.SET_DIAG_LVL_PROT		(0, 12000, 100, eDIAG_PROT_MODE.DIAG_PROT);
OUTGROUP2.CONFIG.SET_DIAG_LVL_PROT		(0, 12000, 100, eDIAG_PROT_MODE.DIAG_PROT);

OUTGROUP0.VAR_IN.xValue:=1;
END_ACTION

ACTION config_inputs:
(* Input Mode Configuration *) // FREQ_SENSE_PERIODS.PERIODS_5, ENCODER_RESOLUTION.EVERY_EDGE
(* Frequency Inputs *)
IN0000.CONFIG.MONITOR		(FILTER_INPUT.UNCHANGED);
IN0001.CONFIG.MONITOR		(FILTER_INPUT.UNCHANGED);
IN0002.CONFIG.MONITOR		(FILTER_INPUT.UNCHANGED);
IN0003.CONFIG.MONITOR		(FILTER_INPUT.UNCHANGED);
IN0500.CONFIG.MONITOR		(FILTER_INPUT.UNCHANGED);
IN0501.CONFIG.MONITOR		(FILTER_INPUT.UNCHANGED);
IN0502.CONFIG.MONITOR		(FILTER_INPUT.UNCHANGED);
IN0503.CONFIG.MONITOR		(FILTER_INPUT.UNCHANGED);
(* Multifuntional Inputs *) 
IN0100.CONFIG.IN_DIGITAL_CSI		(FILTER_INPUT.UNCHANGED);
IN0101.CONFIG.IN_CURRENT_CSI	(FILTER_INPUT.UNCHANGED);
IN0102.CONFIG.MONITOR		(FILTER_INPUT.UNCHANGED);
IN0103.CONFIG.MONITOR		(FILTER_INPUT.UNCHANGED);
IN0200.CONFIG.MONITOR		(FILTER_INPUT.UNCHANGED);
IN0201.CONFIG.MONITOR		(FILTER_INPUT.UNCHANGED);
IN0202.CONFIG.MONITOR		(FILTER_INPUT.UNCHANGED);
IN0203.CONFIG.MONITOR		(FILTER_INPUT.UNCHANGED);
                  				
IN0600.CONFIG.MONITOR		(FILTER_INPUT.UNCHANGED);
IN0601.CONFIG.MONITOR		(FILTER_INPUT.UNCHANGED);
IN0602.CONFIG.MONITOR		(FILTER_INPUT.UNCHANGED);
IN0603.CONFIG.MONITOR		(FILTER_INPUT.UNCHANGED);
IN0700.CONFIG.MONITOR		(FILTER_INPUT.UNCHANGED);
IN0701.CONFIG.MONITOR		(FILTER_INPUT.UNCHANGED);
IN0702.CONFIG.MONITOR		(FILTER_INPUT.UNCHANGED);
IN0703.CONFIG.MONITOR		(FILTER_INPUT.UNCHANGED);
(* Digital Inputs *) 				
IN0300.CONFIG.MONITOR		(FILTER_INPUT.UNCHANGED);
IN0301.CONFIG.MONITOR		(FILTER_INPUT.UNCHANGED);
IN0800.CONFIG.MONITOR		(FILTER_INPUT.UNCHANGED);
IN0801.CONFIG.MONITOR		(FILTER_INPUT.UNCHANGED);
(* Resistopr Inputs *)      	
IN0400.CONFIG.MONITOR		(FILTER_INPUT.UNCHANGED);
IN0401.CONFIG.MONITOR		(FILTER_INPUT.UNCHANGED);
IN0900.CONFIG.MONITOR		(FILTER_INPUT.UNCHANGED);
IN0901.CONFIG.MONITOR		(FILTER_INPUT.UNCHANGED);

(* Diagnostic and Protection Configuration *) //eDIAG_PROT_MODE.DIAG_PROT
(* Frequency Inputs *) 
IN0000.CONFIG.SET_DIAG_LVL_PROT		(0, 32000, 100, eDIAG_PROT_MODE.DIAG_PROT);
IN0001.CONFIG.SET_DIAG_LVL_PROT		(0, 32000, 100, eDIAG_PROT_MODE.DIAG_PROT);
IN0002.CONFIG.SET_DIAG_LVL_PROT		(0, 32000, 100, eDIAG_PROT_MODE.DIAG_PROT);
IN0003.CONFIG.SET_DIAG_LVL_PROT		(0, 32000, 100, eDIAG_PROT_MODE.DIAG_PROT);
IN0500.CONFIG.SET_DIAG_LVL_PROT		(0, 32000, 100, eDIAG_PROT_MODE.DIAG_PROT);
IN0501.CONFIG.SET_DIAG_LVL_PROT		(0, 32000, 100, eDIAG_PROT_MODE.DIAG_PROT);
IN0502.CONFIG.SET_DIAG_LVL_PROT		(0, 32000, 100, eDIAG_PROT_MODE.DIAG_PROT);
IN0503.CONFIG.SET_DIAG_LVL_PROT		(0, 32000, 100, eDIAG_PROT_MODE.DIAG_PROT);
(* Multifuntional Inputs *)                          
IN0100.CONFIG.SET_DIAG_LVL_PROT		(0, 32000, 100, eDIAG_PROT_MODE.DIAG_PROT);
IN0101.CONFIG.SET_DIAG_LVL_PROT		(0, 32000, 100, eDIAG_PROT_MODE.DIAG_PROT);
IN0102.CONFIG.SET_DIAG_LVL_PROT		(0, 32000, 100, eDIAG_PROT_MODE.DIAG_PROT);
IN0103.CONFIG.SET_DIAG_LVL_PROT		(0, 32000, 100, eDIAG_PROT_MODE.DIAG_PROT);
IN0200.CONFIG.SET_DIAG_LVL_PROT		(0, 32000, 100, eDIAG_PROT_MODE.DIAG_PROT);
IN0201.CONFIG.SET_DIAG_LVL_PROT		(0, 32000, 100, eDIAG_PROT_MODE.DIAG_PROT);
IN0202.CONFIG.SET_DIAG_LVL_PROT		(0, 32000, 100, eDIAG_PROT_MODE.DIAG_PROT);
IN0203.CONFIG.SET_DIAG_LVL_PROT		(0, 32000, 100, eDIAG_PROT_MODE.DIAG_PROT);
                                                     
IN0600.CONFIG.SET_DIAG_LVL_PROT		(0, 32000, 100, eDIAG_PROT_MODE.DIAG_PROT);
IN0601.CONFIG.SET_DIAG_LVL_PROT		(0, 32000, 100, eDIAG_PROT_MODE.DIAG_PROT);
IN0602.CONFIG.SET_DIAG_LVL_PROT		(0, 32000, 100, eDIAG_PROT_MODE.DIAG_PROT);
IN0603.CONFIG.SET_DIAG_LVL_PROT		(0, 32000, 100, eDIAG_PROT_MODE.DIAG_PROT);
IN0700.CONFIG.SET_DIAG_LVL_PROT		(0, 32000, 100, eDIAG_PROT_MODE.DIAG_PROT);
IN0701.CONFIG.SET_DIAG_LVL_PROT		(0, 32000, 100, eDIAG_PROT_MODE.DIAG_PROT);
IN0702.CONFIG.SET_DIAG_LVL_PROT		(0, 32000, 100, eDIAG_PROT_MODE.DIAG_PROT);
IN0703.CONFIG.SET_DIAG_LVL_PROT		(0, 32000, 100, eDIAG_PROT_MODE.DIAG_PROT);
(* Digital Inputs *)                                 
IN0300.CONFIG.SET_DIAG_LVL_PROT		(0, 32000, 100, eDIAG_PROT_MODE.DIAG_PROT);
IN0301.CONFIG.SET_DIAG_LVL_PROT		(0, 32000, 100, eDIAG_PROT_MODE.DIAG_PROT);
IN0800.CONFIG.SET_DIAG_LVL_PROT		(0, 32000, 100, eDIAG_PROT_MODE.DIAG_PROT);
IN0801.CONFIG.SET_DIAG_LVL_PROT		(0, 32000, 100, eDIAG_PROT_MODE.DIAG_PROT);
(* Resistopr Inputs *)                               
IN0400.CONFIG.SET_DIAG_LVL_PROT		(0, 32000, 100, eDIAG_PROT_MODE.DIAG_PROT);
IN0401.CONFIG.SET_DIAG_LVL_PROT		(0, 32000, 100, eDIAG_PROT_MODE.DIAG_PROT);
IN0900.CONFIG.SET_DIAG_LVL_PROT		(0, 32000, 100, eDIAG_PROT_MODE.DIAG_PROT);
IN0901.CONFIG.SET_DIAG_LVL_PROT		(0, 32000, 100, eDIAG_PROT_MODE.DIAG_PROT);

(* Digital Switching Threshold - Default ON:= 0.7*Vbb, OFF:= 0.3*Vbb *)
(* Frequency Inputs *)
IN0000.CONFIG.SET_SWITCH_THRESHOLD(300, 700);
IN0001.CONFIG.SET_SWITCH_THRESHOLD(300, 700);
IN0002.CONFIG.SET_SWITCH_THRESHOLD(300, 700);
IN0003.CONFIG.SET_SWITCH_THRESHOLD(300, 700);
IN0500.CONFIG.SET_SWITCH_THRESHOLD(300, 700);
IN0501.CONFIG.SET_SWITCH_THRESHOLD(300, 700);
IN0502.CONFIG.SET_SWITCH_THRESHOLD(300, 700);
IN0503.CONFIG.SET_SWITCH_THRESHOLD(300, 700);
(* Multifuntional Inputs *) 
IN0100.CONFIG.SET_SWITCH_THRESHOLD(300, 700);
IN0101.CONFIG.SET_SWITCH_THRESHOLD(300, 700);
IN0102.CONFIG.SET_SWITCH_THRESHOLD(300, 700);
IN0103.CONFIG.SET_SWITCH_THRESHOLD(300, 700);
IN0200.CONFIG.SET_SWITCH_THRESHOLD(300, 700);
IN0201.CONFIG.SET_SWITCH_THRESHOLD(300, 700);
IN0202.CONFIG.SET_SWITCH_THRESHOLD(300, 700);
IN0203.CONFIG.SET_SWITCH_THRESHOLD(300, 700);
      
IN0600.CONFIG.SET_SWITCH_THRESHOLD(300, 700);
IN0601.CONFIG.SET_SWITCH_THRESHOLD(300, 700);
IN0602.CONFIG.SET_SWITCH_THRESHOLD(300, 700);
IN0603.CONFIG.SET_SWITCH_THRESHOLD(300, 700);
IN0700.CONFIG.SET_SWITCH_THRESHOLD(300, 700);
IN0701.CONFIG.SET_SWITCH_THRESHOLD(300, 700);
IN0702.CONFIG.SET_SWITCH_THRESHOLD(300, 700);
IN0703.CONFIG.SET_SWITCH_THRESHOLD(300, 700);
(* Digital Inputs *)  
IN0300.CONFIG.SET_SWITCH_THRESHOLD(300, 700);
IN0301.CONFIG.SET_SWITCH_THRESHOLD(300, 700);
IN0800.CONFIG.SET_SWITCH_THRESHOLD(300, 700);
IN0801.CONFIG.SET_SWITCH_THRESHOLD(300, 700);
(* Resistopr Inputs *)   
IN0400.CONFIG.SET_SWITCH_THRESHOLD(300, 700);
IN0401.CONFIG.SET_SWITCH_THRESHOLD(300, 700);
IN0900.CONFIG.SET_SWITCH_THRESHOLD(300, 700);
IN0901.CONFIG.SET_SWITCH_THRESHOLD(300, 700);
END_ACTION

END_PROGRAM

// StandardPLC/Application/Temp_Logic
PROGRAM Temp_Logic
VAR
	rawAnalogTemp : INT;         // From temperature analog input
	 // --- Outputs / Display ---
    Temperature_Celsius : REAL;  // Real temperature in °C
    
    Rounded_Temp        : INT;   // Integer value for HMI display

    // --- Control ---
    xDrive      : BOOL;
    uiSpeed     : UINT := 500;
    uiFrequency : UINT;
    uiValue     : UINT;
    xDirection  : BOOL := TRUE;
    xReset      : BOOL := FALSE;
	xEnable: INT;
END_VAR

IOWrapper.READ_INPUTS();

OUTGROUP0.VAR_IN.xValue := TRUE;
// === INPUT READ ===
IOWrapper.READ_INPUTS();

rawAnalogTemp := IN0101.VAR_OUT.uiValueAnalogue;
inc1.array1[2] := PLC_PRG.rawAnalogTemp ;

// === TEMPERATURE CONVERSION (0–25000 raw = –50 to 150°C) ===
Temperature_Celsius := (rawAnalogTemp) * 200.0 / 27000.0 - 50.0;
Rounded_Temp := REAL_TO_INT(Temperature_Celsius); // ✅ Correct




// === MOTOR CONTROL (Trigger at > 60°C) ===
IF rawAnalogTemp > 10800 THEN // (60°C = ((60 + 50) / 200) * 25000)
    xDrive := TRUE;
ELSE
    xDrive := FALSE;
END_IF

IF xDrive THEN
    uiFrequency := uiSpeed;
    uiValue := uiSpeed;
ELSE
    uiFrequency := 0;
    uiValue := 0;
END_IF

// === MOTOR OUTPUT ===
OUT0006.VAR_IN.uiBrakeValue := 0;
OUT0006.VAR_IN.uiValue := uiValue;
OUT0006.VAR_IN.xDirection := xDirection;
OUT0006.VAR_IN.xResetError := xReset;
IOWrapper.WRITE_OUTPUTS();

END_PROGRAM

// StandardPLC/Application/CAN_INIT
PROGRAM CAN_INIT
VAR
		xInit: BOOL:= TRUE;
	
	CAN1_Enable: ifmRCAN.CAN_Enable;
END_VAR

	IF xInit THEN
		CAN1_Enable(
	xEnable:= TRUE,
	eChannel:= ifmDevice.CHAN_1,
	eBaudrate:= ifmDevice.KBAUD_250);
	xInit:= FALSE;	
	END_IF

END_PROGRAM

// StandardPLC/Application/CAN_TX
PROGRAM CAN_TX
VAR
		CAN_TX: ifmRCAN.CAN_TX;
	CANStatus:ifmRCAN.CAN_Status;
	aDATA: ARRAY[0..7] OF USINT:=[1,1,1,2,5,11,0,1];
	
	
	TON_1: TON;
	
	TON0: TON;
	Q: BOOL;
	CAN_Status_0: ifmRCAN.CAN_Status;
	xEnable: BOOL := FALSE;
	TON1: BOOL;
END_VAR

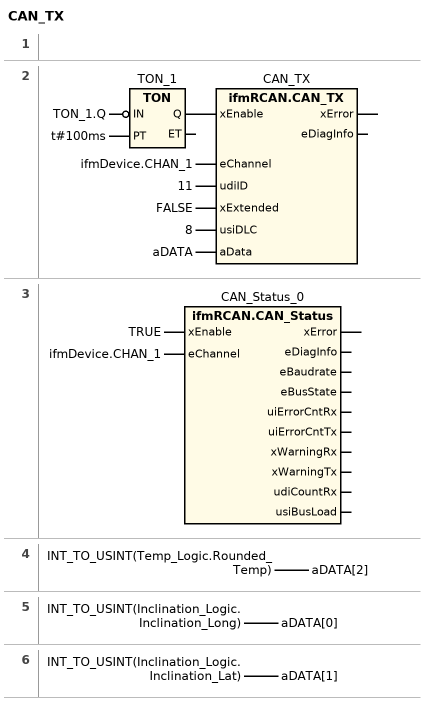
// NETWORK 1

// NETWORK 2
TON_1(IN := NOT TON_1.Q, PT := t#100ms); // TON
CAN_TX(
    xEnable := TON_1.Q,
    eChannel := ifmDevice.CHAN_1,
    udiID := 11,
    xExtended := FALSE,
    usiDLC := 8,
    aData := aDATA); // ifmRCAN.CAN_TX

// NETWORK 3
CAN_Status_0(xEnable := TRUE, eChannel := ifmDevice.CHAN_1); // ifmRCAN.CAN_Status

// NETWORK 4
aDATA[2] := INT_TO_USINT(Temp_Logic.Rounded_Temp);

// NETWORK 5
aDATA[0] := INT_TO_USINT(Inclination_Logic.Inclination_Long);

// NETWORK 6
aDATA[1] := INT_TO_USINT(Inclination_Logic.Inclination_Lat);

END_PROGRAM

// StandardPLC/Application/Inclination_logic
PROGRAM Inclination_logic
VAR

	iSlopeLat: INT;
	iSlopeLong: INT;
	Inclination_Long: INT;
	Inclination_Lat: INT;
END_VAR

// === INPUT READ ===
IOWrapper.READ_INPUTS();
inc1.array1[1] := PLC_PRG.iSlopeLong;	
inc1.array1[0] := PLC_PRG.iSlopeLat;

OUTGROUP0.VAR_IN.xValue := TRUE;

// === INCLINATION CONVERSION (0–65535 = 0°–360°) ===
Inclination_Lat := REAL_TO_INT((PLC_PRG.iSlopeLat) * 360.0 / 65535.0);
Inclination_Long := REAL_TO_INT((PLC_PRG.iSlopeLong) * 360.0 / 65535.0);



// === LED CONTROL BASED ON Inclination_Long ===
IF Inclination_Long < 11.0 THEN
    OUT0001.VAR_IN.uiValue := 1;  // GREEN ON
    OUT0002.VAR_IN.uiValue := 0;  // BLUE OFF
    OUT0003.VAR_IN.uiValue := 0;  // RED OFF

ELSIF Inclination_Long < 16.0 THEN
    OUT0001.VAR_IN.uiValue := 0;  // GREEN OFF
    OUT0002.VAR_IN.uiValue := 1;  // BLUE ON
    OUT0003.VAR_IN.uiValue := 0;  // RED OFF

ELSE
    OUT0001.VAR_IN.uiValue := 0;  // GREEN OFF
    OUT0002.VAR_IN.uiValue := 0;  // BLUE OFF
    OUT0003.VAR_IN.uiValue := 1;  // RED ON
END_IF


// === WRITE OUTPUTS ===
IOWrapper.WRITE_OUTPUTS();

END_PROGRAM

// StandardPLC/Application/test
PROGRAM test 
VAR
	LIN_TRAFO_0: LIN_TRAFO;
END_VAR

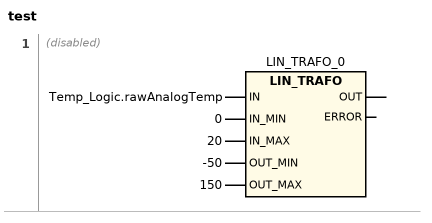
// NETWORK 1 (disabled)
// LIN_TRAFO_0(IN := Temp_Logic.rawAnalogTemp, IN_MIN := 0, IN_MAX := 20, OUT_MIN := -50, OUT_MAX := 150); // LIN_TRAFO

END_PROGRAM

// StandardPLC/Application/Visualization
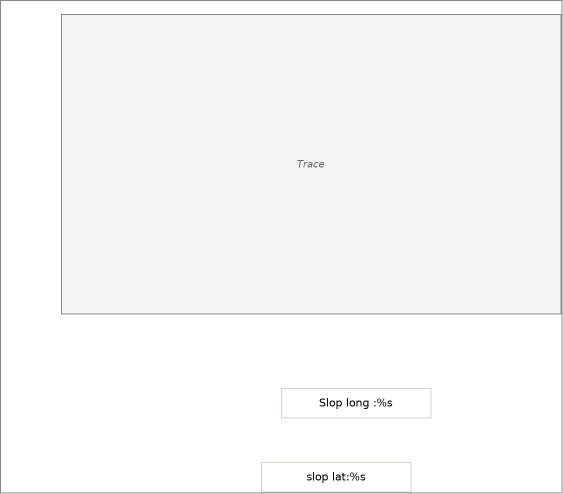
VISUALIZATION Visualization  // 563x494
    Trace (61,14 500x300)
    Textfield (281,388 150x30), "Slop long :%s", text variable: PLC_PRG.iSlopeLong
    Textfield (261,462 150x30), "slop lat:%s"
END_VISUALIZATION

// StandardPLC/Application/Visualization_1
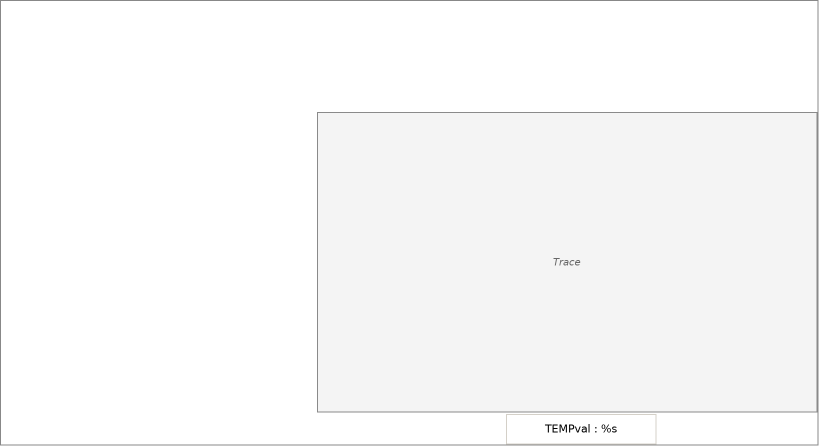
VISUALIZATION Visualization_1  // 819x446
    Trace (317,112 500x300)
    Textfield (506,414 150x30), "TEMPval : %s"
END_VISUALIZATION
